FUNCTION FC_SCALE : REAL
VAR_INPUT
	In : REAL;
	Conf : TYP_SCALE_CONF;
END_VAR
VAR
END_VAR

FC_SCALE := ((Conf.OutMax - Conf.OutMin) / (Conf.InMax - Conf.InMin) * In) + Conf.OutMin;

END_FUNCTION

(* stored: Version 1.1.0.1, ProductVersion 3.1.4024.12
   POU FC_SCALE: Id {5436500b-12cc-4fe8-bf79-dc16f19ace2d}, SpecialFunc None *)
